FUNCTION SCALE_ESC (* Scaling Function Block with escape *)
  (* Standard: 61499-1; Description: Copyright (c) 2024 HR Agrartechnik GmbH This program and the accompanying materials are made available under the terms of the Eclipse Public License 2.0 which is available at https://www.eclipse.org/legal/epl-2.0/ SPDX-License-Identifier: EPL-2.0 *)
  (* Version 1.0, 2024-09-19, Franz Höpfinger, HR Agrartechnik GmbH *)
  PACKAGE signalprocessing;
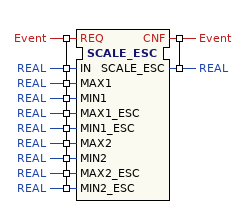
  EVENT_INPUT
    REQ WITH IN, MAX1, MIN1, MAX1_ESC, MIN1_ESC, MAX2, MIN2, MAX2_ESC, MIN2_ESC;
  END_EVENT
  EVENT_OUTPUT
    CNF WITH SCALE_ESC;
  END_EVENT
  VAR_INPUT
    IN : REAL;
    MAX1 : REAL; (* Maximum Input *)
    MIN1 : REAL; (* Minimum Input *)
    MAX1_ESC : REAL; (* Maximum Input Escape, if IN is bigger, Output is MAX2_ESC *)
    MIN1_ESC : REAL; (* Minimum Input Escape, if IN is smaller, Output is MIN2_ESC *)
    MAX2 : REAL; (* Maximum Ouput *)
    MIN2 : REAL; (* Minimum Output *)
    MAX2_ESC : REAL; (* Maximum Ouput Escape *)
    MIN2_ESC : REAL; (* Minimum Output Escape *)
  END_VAR
  VAR_OUTPUT
    SCALE_ESC : REAL;
  END_VAR
  BODY IN ST:
PACKAGE signalprocessing;

(* Scaling Function Block with escape *)
FUNCTION SCALE_ESC : REAL
VAR_INPUT
	IN : REAL;
	MAX1 : REAL;    // Maximum Input
	MIN1 : REAL;    // Minimum Input
	MAX1_ESC : REAL;    // Maximum Input Escape, if IN is bigger, Output is MAX2_ESC
	MIN1_ESC : REAL;    // Minimum Input Escape, if IN is smaller, Output is MIN2_ESC
	MAX2 : REAL;    // Maximum Ouput
	MIN2 : REAL;    // Minimum Output
	MAX2_ESC : REAL;    // Maximum Ouput Escape
	MIN2_ESC : REAL;    // Minimum Output Escape
END_VAR

IF (IN < MIN1_ESC) THEN
	SCALE_ESC := MIN2_ESC;
ELSIF (IN > MAX1_ESC) THEN
	SCALE_ESC := MAX2_ESC;
ELSE
	SCALE_ESC := (IN - MIN1) * (MAX2 - MIN2) / (MAX1 - MIN1) + MIN2;
END_IF;

END_FUNCTION
  END_BODY
END_FUNCTION
